{attribute addProperty BoxType "AX5206-0000-0200-0200"}
{attribute addProperty Id "Drive_status_wordAT %I*UINT1620Position_feedback_1_valueAT %I*DINT3240Following_distanceAT %I*DINT3240"}
{attribute addProperty CRC "368878502"}
{attribute addProperty SizeInBites "80"}
{attribute addProperty SizeInBytes "10"}
TYPE AT_15FCA3A6 :
STRUCT
	{attribute addProperty Name "Drive_status_word"}
	Drive_status_word AT %I* : UINT;
	{attribute addProperty Name "Position_feedback_1_value"}
	Position_feedback_1_value AT %I* : DINT;
	{attribute addProperty Name "Following_distance"}
	Following_distance AT %I* : DINT;
END_STRUCT
END_TYPE

(* stored: Version 1.2.0.0, ProductVersion 3.1.4024.9
   DUT AT_15FCA3A6: Id {b7d289b9-e602-4814-ad6c-72df6e53093f} *)
